INTERFACE ITF_GroupE_TE1_HMI_Connector EXTENDS ITF_BaseGroupElement_HMI_Connector

END_INTERFACE

(* stored: Version 1.1.0.1, ProductVersion 3.1.4024.15
   Itf ITF_GroupE_TE1_HMI_Connector: Id {f7956722-b5fa-4e37-83b9-9d572c084144} *)
